{attribute 'qualified_only'}
VAR_GLOBAL
END_VAR

VAR_GLOBAL CONSTANT
    nESTOP_NUM: UINT := 2;
	nLIGHTCURTAIN_NUM : UINT :=2;
	nSAFETYZONE_NUM : UINT :=2;
END_VAR

(* stored: Version 1.1.0.1, ProductVersion 3.1.4024.13
   GVL GVL_SAFETY: Id {fe1476ef-6e5a-45ac-b16c-b9bd22946e99} *)
